// TIA Portal project "variantPointerProject" (V16)

(* hardware
DEVICE "S71500/ET200MP station_1"  S7-1500 station
   slot 0: "Rail_0"  Rack  6ES7 590-1***0-0AA0
   slot 1: "PLC_2"  CPU 1511-1 PN  6ES7 511-1AK02-0AB0  V2.8
      slot 3: "CPU display_1"  6ES7591-1AA00-0AA0
      slot 32768: "PROFINET interface_1"  X1
         slot 32769: "Port_1"  X1 P1
         slot 32770: "Port_2"  X1 P2
      slot 34817: "Virtual CP interface port_1"  Virtual CP interface port  Virtual CP interface port
*)

// ===== PLC "PLC_2"  CPU 1511-1 PN =====

TYPE "TCircle"
   STRUCT
      Radius : Real;   // The radius of circle
      Area : Real;   // Area of Circle
   END_STRUCT;
END_TYPE

TYPE "TRectangle"
   STRUCT
      Height : Real;   // Height of Rectangle
      Base : Real;   // Base of rectangle
      Area : Real;   // Area of Rectangle
   END_STRUCT;
END_TYPE

TYPE "TTriangle"
   STRUCT
      Height : Real;   // height of triangle
      Base : Real;   // base of triangle
      Area : Real;   // area of triangle
   END_STRUCT;
END_TYPE

DATA_BLOCK "shapes"   // DB1
{ S7_Optimized_Access := 'TRUE' }
VERSION : 0.1
   VAR
      triangle : "TTriangle";
      circle : "TCircle";
      rectangle : "TRectangle";
      triangleArea : Real;
      circleArea : Real;
      rectangleArea : Real;
   END_VAR
BEGIN
END_DATA_BLOCK

FUNCTION "CalcArea" : Real   // FC1, SCL
{ S7_Optimized_Access := 'TRUE' }
VERSION : 0.1
   VAR_IN_OUT
      Object : Variant;
   END_VAR
   VAR_TEMP
      TmpCircle : REF_TO "TCircle";
      TmpRectangle : REF_TO "TRectangle";
      TmpTriangle : REF_TO "TTriangle";
      tempResult : Real;
   END_VAR
   VAR CONSTANT
      CF_PI : Real := 3.141593;   // PI Value
   END_VAR
BEGIN


   CASE TypeOf(#Object) OF
       TCircle:
           #TmpCircle ?= #Object;
           IF #TmpCircle <> NULL THEN
               #CalcArea := #TmpCircle<?OpDeref?>.Area := #TmpCircle<?OpDeref?>.Radius ** 2 * #CF_PI;//use ** operator for power of a number
               #tempResult := #CalcArea;

           END_IF;
       TRectangle:
           #TmpRectangle ?= #Object;
           IF #TmpRectangle <> null THEN
               #CalcArea := #TmpRectangle<?OpDeref?>.Area := #TmpRectangle<?OpDeref?>.Height * #TmpRectangle<?OpDeref?>.Base;
               #tempResult := #CalcArea;

           END_IF;
       TTriangle:
           #TmpTriangle ?= #Object;
           IF #TmpTriangle <> NULL THEN
               #CalcArea := #TmpTriangle<?OpDeref?>.Area := (#TmpTriangle<?OpDeref?>.Height * #TmpTriangle<?OpDeref?>.Base) / 2.0;
               #tempResult := #CalcArea;

           END_IF;
       ELSE  
           #tempResult := 0.0;

   END_CASE;

   #CalcArea := #tempResult;
END_FUNCTION

ORGANIZATION_BLOCK "Main"   // OB1, LAD, ProgramCycle
TITLE = "Main Program Sweep (Cycle)"
{ S7_Optimized_Access := 'TRUE' }
VERSION : 0.1
   VAR_INPUT
      Initial_Call : Bool;   // Initial call of this OB
      Remanence : Bool;   // =True, if remanent data are available
   END_VAR
BEGIN

REGION Network 2 (SCL)
   "shapes".rectangleArea := "CalcArea"("shapes".rectangle);
   "shapes".triangleArea := "CalcArea"("shapes".triangle);
   "shapes".circleArea := "CalcArea"("shapes".circle);
END_REGION
END_ORGANIZATION_BLOCK